Staubli VAL3: chinese.dtx

mdesc mNomSpeed
string sValProduct
